Staubli VAL3: robotMove.pjx

--- robotMove.pjx ---
Parameters version=s7.9.1 stackSize=5000 millimeterUnit=true
Program file=robotMove.pgx
Program file=start.pgx
Program file=stop.pgx
Data file=robotMove.dtx
Type name=JointSpace path=Disk://RobotController_Libs/RobotStatus/JointSpace/JointSpace.pjx
Type name=FlagStatus path=Disk://RobotController_Libs/FlagStatus/FlagStatus.pjx

--- robotMove.pgx ---
public program robotMove(FlagStatus& x_fFlagStatus, JointSpace& x_jMoveCommand)
begin

  //This program is used for realtime robot control, and it should be called every 4ms(standard robot loop time).
  //It will move the robot to the given goal position based on the current judging condition(robot condition and
  //contact force) in every 4ms. And the program will keep the current judging condition interface reserved for
  //future function expansion.

  //Judge the current host ROS command, robot status and contact force and then decide whether the loop will begin.
  while (x_fFlagStatus.RosFlag==1 and x_fFlagStatus.RobotFlag==1 and x_fFlagStatus.ForceFlag==1)

    //Send the joint command for the next 4ms, and returns true if command accepted, false if refuesed.(movejSync
    //instruction not started or already completed.)
    if(!$movejSync(x_jMoveCommand.JointPos))
      popUpMsg("The joint motion command refused and robot will stop.")
      return
    endIf

    //Force the sequencing to the next task by using the "delay(0.0)" instruction explicitly.
    delay(0.0)

  endWhile

  //End the Sychronous Movej procedural motion mode and stop the robot.
  $movejSyncEnd()
  stopMove()

end
